TYPE csp_transfer_upstacker_connection_status_enum :
(		
	CSP_TRANSFER_UPSTACKER_STATUS_CONNECTION_START							:= 0,
	CSP_TRANSFER_UPSTACKER_STATUS_CONNECTION_ENGAGE							:= 10,
	CSP_TRANSFER_UPSTACKER_STATUS_CONNECTION_ENGAGED						:= 20,
	CSP_TRANSFER_UPSTACKER_STATUS_CONNECTION_CHECK_CHANGE_CAM				:= 30,
	CSP_TRANSFER_UPSTACKER_STATUS_CONNECTION_CHANGE_CAM						:= 40,
	CSP_TRANSFER_UPSTACKER_STATUS_CONNECTION_WAIT_NEW_CAM					:= 50,
	CSP_TRANSFER_UPSTACKER_STATUS_CONNECTION_DONE 							:= 900,
	CSP_TRANSFER_UPSTACKER_STATUS_CONNECTION_ERROR 							:= 999
) := CSP_TRANSFER_UPSTACKER_STATUS_CONNECTION_START;
END_TYPE

(* stored: Version 1.1.0.1, ProductVersion 3.1.4022.12
   DUT csp_transfer_upstacker_connection_status_enum: Id {e6898b8a-7110-47f5-87e4-5c10658b6f6f} *)
